FUNCTION_BLOCK TrueBoolValue IMPLEMENTS BoolValue
VAR
END_VAR

{attribute 'monitoring' := 'call'}
PROPERTY Value : BOOL
GET
Value := TRUE;
END_GET
END_PROPERTY

END_FUNCTION_BLOCK

(* stored: Version 1.1.0.1
   POU TrueBoolValue: Id {32544c48-7ac0-4545-b8e7-eec2336e8f9e}, SpecialFunc None
   Property Value: Id {466e9ca4-1de8-43d8-8bec-ef7297ae9bf7}
   Get Get: Id {53b48b8a-4560-499f-8562-2f221b611a10} *)
